Universal Robots PolyScope program: swan2.urp

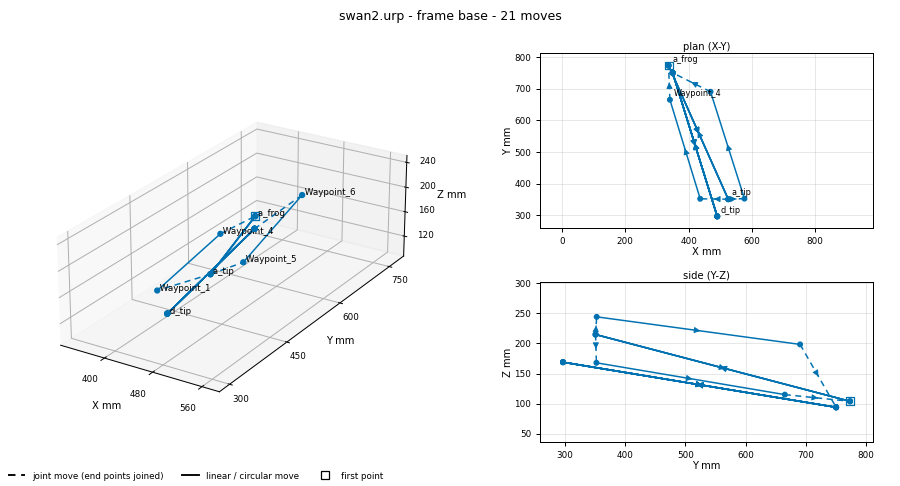
[picture p0: tool path of swan2.urp in frame base, 21 of 21 moves have a stored position in this frame; points joined in program order, loops and branches not executed]
Program swan2 (installation=string_planes directory=/programs createdIn=5.17.3 lastSavedIn=5.17.3 robotSerialNumber=20245501435)
Calibrated DH parameters: a=[0.000154, -0.137004, -0.385524, -0.00002, 0.000092, 0]; d=[0.162441, 211.794786, -230.585024, 18.923638, 0.099786, 0.09951]; alpha=[1.569493, -0.001902, 0.003874, 1.570111, -1.570167, 0]; deltaTheta=[0, -1.242934, 1.056292, 0.186646, 0.000002, 0.000001]
InitVariablesNode
Robot Program (runOnlyOnce=false)
  Call Swan
SubProgram -> Swan
SubProgram Swan (keepSynchronizedWithDisk=false) programFile=/programs/Swan.urp
  Timer (action=Start) variable(name=beats)
  MoveL speed 150 mm/s, acceleration 600 mm/s^2 (useActiveTCP=true) feature=Base
    Waypoint a_frog: TCP in base x=336.638 y=773.336 z=103.937 mm, rx=-1.3698 ry=-2.3362 rz=1.327 rad; joints [-127.102, -6.181, 18.995, -50.118, -88.699, -156.884] deg; TCP offset x=28.21 y=-96.107 z=-99.69 mm, rx=0 ry=0 rz=0 rad
    Waypoint a_tip: TCP in base x=525.206 y=350.983 z=214.78 mm, rx=-1.3698 ry=-2.3362 rz=1.327 rad; joints [-161.028, -44.56, 81.191, -78.693, -115.03, -178.818] deg
      Until EXPRESSION (allowActions=false) ExpressionBranch=beats≥3
    Timer (action=Reset) variable=beats
  MoveJ speed 60 deg/s, acceleration 80 deg/s^2 (useActiveTCP=true) feature=Base
    Waypoint Waypoint_1: motionParameters(blendRadius=0.03); TCP in base x=436.609 y=352.375 z=167.842 mm, rx=-1.4774 ry=-2.3156 rz=1.0625 rad; joints [-158.188, -47.761, 97.715, -98.035, -103.646, -177.64] deg
  Timer (action=Reset) variable=beats
  MoveL speed 150 mm/s, acceleration 500 mm/s^2 (useActiveTCP=true) feature=Base
    Waypoint Waypoint_4: TCP in base x=340.943 y=665.128 z=115.023 mm, rx=-1.4671 ry=-2.3126 rz=0.9695 rad; joints [-132.154, -25.951, 61.091, -84.349, -83.311, -159.675] deg
      Until EXPRESSION (allowActions=false) ExpressionBranch=beats≥3
  MoveJ speed 60 deg/s, acceleration 80 deg/s^2 (useActiveTCP=true) feature=Base
    Waypoint a_frog: TCP in base x=336.638 y=773.336 z=103.937 mm, rx=-1.3698 ry=-2.3362 rz=1.327 rad; joints [-127.102, -6.181, 18.995, -50.118, -88.699, -156.884] deg
  Timer (action=Reset) variable=beats
  MoveL speed 100 mm/s, acceleration 300 mm/s^2 (useActiveTCP=true) feature=Base
    Waypoint a_tip: motionParameters(blendRadius=0.03); TCP in base x=525.206 y=350.983 z=214.78 mm, rx=-1.3698 ry=-2.3362 rz=1.327 rad; joints [-161.028, -44.56, 81.191, -78.693, -115.03, -178.818] deg
      Until EXPRESSION (allowActions=false) ExpressionBranch=beats≥2.5
  Timer (action=Reset) variable=beats
  MoveL speed 300 mm/s, acceleration 1200 mm/s^2 (useActiveTCP=true) feature=Base
    Waypoint a_frog: TCP in base x=336.638 y=773.336 z=103.937 mm, rx=-1.3698 ry=-2.3362 rz=1.327 rad; joints [-127.102, -6.181, 18.995, -50.118, -88.699, -156.884] deg
      Until EXPRESSION (allowActions=false) ExpressionBranch=beats≥0.5
  Timer (action=Reset) variable=beats
  MoveL speed 100 mm/s, acceleration 600 mm/s^2 (useActiveTCP=true) feature=Base
    Waypoint a_tip: motionParameters(blendRadius=0.03); TCP in base x=525.206 y=350.983 z=214.78 mm, rx=-1.3698 ry=-2.3362 rz=1.327 rad; joints [-161.028, -44.56, 81.191, -78.693, -115.03, -178.818] deg
      Until EXPRESSION (allowActions=false) ExpressionBranch=beats≥2
  MoveJ speed 60 deg/s, acceleration 80 deg/s^2 (useActiveTCP=true) feature=Base
    Waypoint Waypoint_5: TCP in base x=576.416 y=352.811 z=244.122 mm, rx=-1.3698 ry=-2.3362 rz=1.327 rad; joints [-162.2, -41.352, 69.945, -71.043, -115.912, -179.715] deg
  MoveL speed 400 mm/s, acceleration 1200 mm/s^2 (useActiveTCP=true) feature=Base
    Waypoint Waypoint_6: TCP in base x=469.305 y=690.432 z=198.38 mm, rx=-1.3698 ry=-2.3362 rz=1.327 rad; joints [-137.273, -11.027, 15.189, -41.782, -96.797, -163.098] deg
  MoveJ speed 60 deg/s, acceleration 80 deg/s^2 (useActiveTCP=true) feature=Base
    Waypoint d_frog: TCP in base x=349.663 y=750.266 z=93.98 mm, rx=-1.41 ry=-2.1761 rz=1.1503 rad; joints [-128.619, -11.447, 33.081, -61.83, -78.179, -158.113] deg
  Timer (action=Reset) variable=beats
  MoveL speed 150 mm/s, acceleration 600 mm/s^2 (useActiveTCP=true) feature=Base
    Waypoint d_tip: TCP in base x=490.401 y=296.853 z=168.858 mm, rx=-1.3783 ry=-2.2079 rz=1.1619 rad; joints [-164.642, -46.076, 94.437, -89.854, -107.25, -182.664] deg
      Until EXPRESSION (allowActions=false) ExpressionBranch=beats≥2
  Timer (action=Reset) variable=beats
  Timer (action=Start) variable=beats
  MoveL speed 150 mm/s, acceleration 600 mm/s^2 (useActiveTCP=true) feature=Base
    Waypoint d_frog: TCP in base x=349.663 y=750.266 z=93.98 mm, rx=-1.41 ry=-2.1761 rz=1.1503 rad; joints [-128.619, -11.447, 33.081, -61.83, -78.179, -158.113] deg
      Until EXPRESSION (allowActions=false) ExpressionBranch=beats≥0.5
  Timer (action=Reset) variable=beats
  MoveL speed 150 mm/s, acceleration 600 mm/s^2 (useActiveTCP=true) feature=Base
    Waypoint d_tip: TCP in base x=490.401 y=296.853 z=168.858 mm, rx=-1.3783 ry=-2.2079 rz=1.1619 rad; joints [-164.642, -46.076, 94.437, -89.854, -107.25, -182.664] deg
      Until EXPRESSION (allowActions=false) ExpressionBranch=beats≥0.5
  Timer (action=Reset) variable=beats
  MoveL speed 150 mm/s, acceleration 600 mm/s^2 (useActiveTCP=true) feature=Base
    Waypoint d_frog: TCP in base x=349.663 y=750.266 z=93.98 mm, rx=-1.41 ry=-2.1761 rz=1.1503 rad; joints [-128.619, -11.447, 33.081, -61.83, -78.179, -158.113] deg
      Until EXPRESSION (allowActions=false) ExpressionBranch=beats≥0.5
  Timer (action=Reset) variable=beats
  MoveL speed 150 mm/s, acceleration 600 mm/s^2 (useActiveTCP=true) feature=Base
    Waypoint d_tip: TCP in base x=490.401 y=296.853 z=168.858 mm, rx=-1.3783 ry=-2.2079 rz=1.1619 rad; joints [-164.642, -46.076, 94.437, -89.854, -107.25, -182.664] deg
      Until EXPRESSION (allowActions=false) ExpressionBranch=beats≥0.5
  Timer (action=Reset) variable=beats
  MoveL speed 150 mm/s, acceleration 600 mm/s^2 (useActiveTCP=true) feature=Base
    Waypoint d_frog: TCP in base x=349.663 y=750.266 z=93.98 mm, rx=-1.41 ry=-2.1761 rz=1.1503 rad; joints [-128.619, -11.447, 33.081, -61.83, -78.179, -158.113] deg
      Until EXPRESSION (allowActions=false) ExpressionBranch=beats≥0.5
  Timer (action=Reset) variable=beats
  MoveL speed 150 mm/s, acceleration 600 mm/s^2 (useActiveTCP=true) feature=Base
    Waypoint d_tip: TCP in base x=490.401 y=296.853 z=168.858 mm, rx=-1.3783 ry=-2.2079 rz=1.1619 rad; joints [-164.642, -46.076, 94.437, -89.854, -107.25, -182.664] deg
      Until EXPRESSION (allowActions=false) ExpressionBranch=beats≥0.5
  Timer (action=Reset) variable=beats
  MoveL speed 150 mm/s, acceleration 600 mm/s^2 (useActiveTCP=true) feature=Base
    Waypoint d_frog: TCP in base x=349.663 y=750.266 z=93.98 mm, rx=-1.41 ry=-2.1761 rz=1.1503 rad; joints [-128.619, -11.447, 33.081, -61.83, -78.179, -158.113] deg
      Until EXPRESSION (allowActions=false) ExpressionBranch=beats≥0.5
  Timer (action=Reset) variable=beats
  MoveL speed 150 mm/s, acceleration 600 mm/s^2 (useActiveTCP=true) feature=Base
    Waypoint d_tip: TCP in base x=490.401 y=296.853 z=168.858 mm, rx=-1.3783 ry=-2.2079 rz=1.1619 rad; joints [-164.642, -46.076, 94.437, -89.854, -107.25, -182.664] deg
      Until EXPRESSION (allowActions=false) ExpressionBranch=beats≥0.5
  Timer (action=Reset) variable=beats
  MoveL speed 100 mm/s, acceleration 500 mm/s^2 (useActiveTCP=true) feature=Base
    Waypoint d_frog: TCP in base x=349.663 y=750.266 z=93.98 mm, rx=-1.41 ry=-2.1761 rz=1.1503 rad; joints [-128.619, -11.447, 33.081, -61.83, -78.179, -158.113] deg
      Until EXPRESSION (allowActions=false) ExpressionBranch=beats≥3.5
  Wait Sleep waitTime=500
